FUNCTION_BLOCK FB_HRErrHist
(* v1.10
build up an error history consisting of two arrays and one index.
The index shows the actual array position. The last error id and the count for this id are saved in the arrays.
If an error id is the same as the previous input error the counter is increased. Otherwise the index is increased.
*)
VAR_INPUT
	bEdgeDetect	: BOOL;	(* FALSE: every input(bErr) is processed; TRUE: only rising edge of input is processed *)
END_VAR
VAR_OUTPUT
	nErrSum		: UINT;
	nErrIdx		: UINT; // error list index of last occured error (max. cHistLen)
	aErrList	: ARRAY[1..cHistLen] OF ST_HRErrHist;
END_VAR

VAR
	bNewErr		: BOOL;
	fbErrTrig	: R_TRIG;
END_VAR
VAR CONSTANT
	cHistLen	: UINT := 100;
END_VAR

METHOD AddError
VAR_INPUT
	bErr		: BOOL;
	hrErrCode	: HRESULT;
	sErrSource	: STRING(63);
END_VAR
fbErrTrig(CLK:=bErr);
IF bEdgeDetect THEN
	bNewErr := fbErrTrig.Q;
ELSE
	bNewErr := bErr;
END_IF

IF bNewErr THEN
	nErrSum := nErrSum + 1;
	IF nErrIdx < cHistLen THEN
		IF nErrIdx = 0 THEN
			nErrIdx	:= nErrIdx + 1;
		ELSIF aErrList[nErrIdx].hrErrCode <> hrErrCode OR aErrList[nErrIdx].sErrSource <> sErrSource THEN
			nErrIdx	:= nErrIdx + 1;
		END_IF
		aErrList[nErrIdx].hrErrCode := hrErrCode;
		aErrList[nErrIdx].sErrSource := sErrSource;
		aErrList[nErrIdx].nErrCount := aErrList[nErrIdx].nErrCount + 1;
	END_IF
END_IF
END_METHOD

METHOD Reset
VAR_INPUT
END_VAR
nErrSum := 0;
nErrIdx := 0;
MEMSET(ADR(aErrList),0,SIZEOF(aErrList));
END_METHOD

END_FUNCTION_BLOCK

(* stored: Version 1.1.0.1, ProductVersion 3.1.4024.12
   POU FB_HRErrHist: Id {6bcf72c4-74b8-44f2-b0ca-82b93036056e}, SpecialFunc None
   Method AddError: Id {b9441b7c-4791-4bd3-b687-8b97db1e2d06}
   Method Reset: Id {9ab4bf07-cf63-4423-b4ff-577151910933} *)
